PROGRAM F_FactoryIO_Read_InputRegs
VAR;
	LFB_MBReadInputRegs 	: FB_MBReadInputRegs;
	bBusy: BOOL;
	bError: BOOL;
END_VAR

LFB_MBReadInputRegs(
	sIPAddr := '127.0.0.1',
	nTCPPort := 505,
	nUnitID := 255,
	nQuantity := 8, // Nombre de registres à lire
	nMBAddr := 0,
	cbLength := SIZEOF(GAB_FactoryIO_InputRegs),
	pDestAddr := ADR(GAB_FactoryIO_InputRegs),
	bExecute := TRUE,
	tTimeout := T#1S,
	bBusy => bBusy,
	bError => bError,
	nErrId => ,
	cbRead => ,
 );
 
 
 
 
LFB_MBReadInputRegs(bExecute := FALSE);

END_PROGRAM

(* stored: Version 1.1.0.1, ProductVersion 3.1.4024.11
   POU F_FactoryIO_Read_InputRegs: Id {316264d6-447a-47b0-92be-e80d12f427b3}, SpecialFunc None *)
